// List of UDINTs.
FUNCTION_BLOCK FB_UdintList
VAR
	List : ARRAY[ 0 .. GVL_List.LIST_SIZE - 1 ] OF UDINT; // hold list
	_Count : UDINT := 0; // number of items.
END_VAR

// Add item to list. TRUE if successful. 
METHOD PUBLIC AddItem : BOOL
VAR_INPUT
	Item : UDINT; // item to add.
END_VAR
IF _Count < GVL_List.LIST_SIZE THEN
	List[_Count] := Item; // list is zero indexed, so number of items points at next free space.
	_Count := _Count + 1; 
	AddItem := TRUE;
END_IF
END_METHOD

// Removes all list items
METHOD PUBLIC Clear
MEMSET(ADR(List[0]), 0, SIZEOF(List));
_Count := 0;
END_METHOD

// TRUE if sItem is in FB_List.
METHOD PUBLIC Contains : INT
VAR_INPUT
	Item : UDINT; // Item to check.
END_VAR
VAR
	i : UINT := 0;
END_VAR
Contains := -1;
i := 0;
WHILE ( (Contains < 0) AND (i < _Count) ) DO
	
	Contains := SEL(Item = List[i], Contains, TO_INT(i) ); // if it matches, return the position.
	i := i + 1;
	
END_WHILE
END_METHOD

{attribute 'monitoring' := 'call'}
// Number of items in list.
PROPERTY PUBLIC Count : UDINT
GET
Count := _Count;
END_GET
END_PROPERTY

// Return item in list at index position. Returns empty string if invalid index.
METHOD PUBLIC GetIndex : UDINT
VAR_INPUT
	Index : UDINT;
END_VAR
THIS^.TryGetIndex(Index,  GetIndex);
END_METHOD

//Remove the specified index. Shuffle remaining so list is intact.
METHOD PUBLIC RemoveIndex : BOOL
VAR_INPUT
	Index : UDINT;
END_VAR
IF Index >= _Count THEN // invalid index request.
	RETURN;
END_IF

IF Index < _Count - 1 THEN // If Index = _Count -1, last two lines sufficient.

	MEMMOVE( 
		destAddr := ADR( List[Index] ), 
		srcAddr := ADR( List[Index + 1] ), 
		n := SIZEOF(List[0]) * (_Count - Index - 1)
	);
	
END_IF

RemoveIndex := TRUE;

List[_Count - 1] := 0; // default the "old" end of the list.
_Count := _Count - 1; // reduce count.
END_METHOD

// TRUE if successful and list item in sItem
METHOD PUBLIC TryGetIndex : BOOL
VAR_INPUT
	Index : UDINT;
END_VAR
VAR_IN_OUT
	Item : UDINT;
END_VAR
IF Index < _Count THEN
	TryGetIndex := TRUE;
	Item := List[Index];
ELSE
	Item := 0;
END_IF
END_METHOD

END_FUNCTION_BLOCK

(* stored: Version 1.1.0.1, ProductVersion 3.1.4020.12
   POU FB_UdintList: Id {61129f84-6c4b-4e65-842c-5f111d53a85c}, SpecialFunc None
   Method AddItem: Id {144122dd-3472-41dd-8536-72f4edb9754c}
   Method Clear: Id {96b68d45-d772-438b-bcc1-9f910df7caf6}
   Method Contains: Id {1e39d79c-d386-48dc-911b-8d9a46fe8290}
   Property Count: Id {de59a019-ec52-488c-9476-616d6f998219}
   Get Get: Id {b9846dd2-e6ee-48d6-bf8b-ac4a751a1efd}
   Method GetIndex: Id {cdd95fd1-cdde-436e-bd15-0f36ccf1c07d}
   Method RemoveIndex: Id {a8897e84-e02c-4c96-9331-58101fc33cdd}
   Method TryGetIndex: Id {366b1afe-3a42-4e19-b655-3354a9151b49} *)
